// TIA Portal V21 export
DATA_BLOCK "CipDo"   // DB202
{ S7_Optimized_Access := 'FALSE' }
// stored: AutoNumber false
   VAR
      MM01CmdMagneticMixerMvCommand : Bool;
      CP01CmdCentrifugalPumpMvAreaCommand : Bool;
      HTR01HooterMvArea : Bool;
      LF01VesselLampOutputMv1000 : Bool;
      SPARE4 : Bool;
      SPARE5 : Bool;
      SPARE6 : Bool;
      SPARE7 : Bool;
   END_VAR
BEGIN
END_DATA_BLOCK
